{attribute 'qualified_only'}
{attribute 'strict'}
TYPE
    State :
    (
        Ready := 0,
        Busy,
        Done,
        Fail
    );
END_TYPE

(* stored: Version 1.1.0.1, ProductVersion 3.1.4024.12
   DUT State: Id {a90331e8-3131-4504-807a-09a9ae7e31d4} *)
